// TwinCAT 3 PLC project Intecre_File
// Title: Intecre.File
// Company: Intecre Ltd
// Author: Mark Lazarides
// ProjectVersion: 1.1.0
// Description: 1.1.0 simplified interface for T_StructurePersistence 1.0.5 Increased JDOC size. 1.0.4 Fixed bug in assigning CSV separator for CsvReader 1.0.3 Clear Read and Write Success flags on struct persistence when req'd.
// ProgramVersion: 3.1.4020.4
// libraries:
//   Intecre.Utilities, * (Intecre Ltd)
//   Tc2_Standard, * (Beckhoff Automation GmbH)
//   Tc2_System, * (Beckhoff Automation GmbH)
//   Tc2_Utilities, * (Beckhoff Automation GmbH)
//   Tc3_JsonXml, * (Beckhoff Automation GmbH)
// project tree:
//   / Character.TcGVL, Param.TcGVL
//   Csv/ T_CsvFileReader.TcPOU, T_CsvFileWriter.TcPOU
//   File Bases/ E_FileBaseStates.TcDUT, T_FileReadBase.TcPOU, T_FileWriteBase.TcPOU
//   GenericFiles/ TxtFileString.TcDUT, T_TxtFileWriter.TcPOU
//   Json/ JsonDoc.TcDUT, JsonParams.TcGVL, T_StructToJsonFileWriter.TcPOU, T_StructFromJsonFileReader.TcPOU
//   Structure Persistence/ E_StructPersistenceStates.TcDUT, ST_PersistenceOptions.TcDUT, T_StructPersistence.TcPOU
//   Utilities/ E_CheckFileExistsStates.TcDUT, T_CheckFileExists.TcPOU
//   Version/ Global_Version.TcGVL

// ---- File Bases/E_FileBaseStates.TcDUT
TYPE E_FileBaseStates :
(
	WaitForStart,
	OpenFile,
	WaitForOpenComplete,
	SeekEnd,
	WaitForSeekEndComplete,
	GetSize,
	WaitForGetSizeComplete,
	SeekStart,
	WaitForSeekStartComplete,
	CreateBuffer,
	ReadFromFile,
	ReadFromFileComplete,
	WriteToFile,
	WriteToFileComplete,
	CloseFile,
	WaitForCloseComplete,
	FinishAndCleanup ) INT := WaitForStart;
END_TYPE

// ---- GenericFiles/TxtFileString.TcDUT
TYPE TxtFileString : STRING(Param.TXT_FILE_MAX_STRING_LENGTH); END_TYPE

// ---- Json/JsonDoc.TcDUT
TYPE JsonDoc : STRING( JsonParams.JSON_DOC_SIZE ); END_TYPE

// ---- Structure Persistence/E_StructPersistenceStates.TcDUT
{attribute 'qualified_only'}
{attribute 'strict'}
TYPE E_StructPersistenceStates :
(
	None,
	Initialise,
	Wait,
	ReadFromFile,
	WaitForReadComplete,
	WriteToFile,
	WaitForWriteComplete,
	Finished
);
END_TYPE

// ---- Structure Persistence/ST_PersistenceOptions.TcDUT
TYPE ST_PersistenceOptions :
STRUCT
	AddressOfStruct : PVOID;
	SizeOfStruct : UDINT;
	NameOfStructureType : STRING; // eg ST_Recipe; NOT the instance name!
	FilePath : STRING; // location to store this
	CreateFileIfDoesntExist : BOOL := TRUE; // if read fails, try a write.
	AutoWriteOnDifference : BOOL := TRUE; // if difference between
	AutoWriteCheckTime : TIME := T#2M; // how often to check for difference
	AutoWriteDebounceTime : TIME := T#30S; // time since last change to write file
END_STRUCT
END_TYPE

// ---- Utilities/E_CheckFileExistsStates.TcDUT
{attribute 'qualified_only'}
{attribute 'strict'}
TYPE E_CheckFileExistsStates :
(	
	WaitForStart,
	WaitForOpenResult,
	CloseIfOpened
);
END_TYPE

// ---- Character.TcGVL
VAR_GLOBAL CONSTANT
	CARRIAGE_RETURN : BYTE := 16#D;
	LINE_FEED : BYTE := 16#A;
	ASCI_SEMI_COLON : BYTE := 16#3B;
	ASCI_COMMA		: BYTE := 16#2C;
END_VAR

// ---- Json/JsonParams.TcGVL
{attribute 'qualified_only'}
VAR_GLOBAL CONSTANT
	JSON_DOC_SIZE : UDINT := 10000; // make this large enough for your largest structure. Add at least 20% to the byte size to account for json syntax.
END_VAR

// ---- Param.TcGVL
{attribute 'qualified_only'}
VAR_GLOBAL CONSTANT
	TXT_FILE_MAX_STRING_LENGTH : UDINT := 300;
END_VAR

// ---- Version/Global_Version.TcGVL
{attribute 'TcGenerated'}
{attribute 'no-analysis'}
{attribute 'linkalways'}
// This function has been automatically generated from the project information.
VAR_GLOBAL CONSTANT
	{attribute 'const_non_replaced'}
	stLibVersion_Intecre_File : ST_LibVersion := (iMajor := 1, iMinor := 1, iBuild := 0, iRevision := 0, nFlags := 0, sVersion := '1.1.0');
END_VAR

// ---- Csv/T_CsvFileReader.TcPOU
// Usage:
// Call instance (i.e. ofbCsvRead();) every scan while waiting for operations to complete.
// SetFileParams() Set the File directory and separator variable. 
// GetFile() Get the File.
// #various props: Observe the properties to see whether it passed the file checks.
// NextField() Next through the fields of the CSV. 
// #sField, Row, Column: Use properties to access values, using row and column.
FUNCTION_BLOCK T_CsvFileReader
VAR
// state vars.
	filePath : Tc2_Utilities.T_MaxString; // filepath
	firstField : BOOL;
	newRow : BOOL;
	
// backing properties	
	_Row : UINT;(* Row number (record) *)
	_Column : UINT;(* Column number (record field) *)
	_Field : Tc2_Utilities.T_MaxString; // Field in current Row and column
	
// Objects	
	fileRead : T_FileReadBase;(* Writes one record (line) *)
	csvReader : Tc2_Utilities.FB_CSVMemBufferReader; // read bits
	
END_VAR

fileRead();

{attribute 'monitoring' := 'call'}
PROPERTY PUBLIC Busy : BOOL
GET
Busy := fileRead.Busy;
END_GET
END_PROPERTY

PROPERTY PUBLIC Column : UINT
GET
Column := _Column;
END_GET
END_PROPERTY

{attribute 'monitoring' := 'call'}
PROPERTY PUBLIC Eof : BOOL
GET
Eof := ReadyForParsing AND NOT csvReader.bOk AND NOT firstField;
END_GET
END_PROPERTY

{attribute 'monitoring' := 'call'}
PROPERTY PUBLIC Error : BOOL
GET
Error := fileRead.Error;
END_GET
END_PROPERTY

{attribute 'monitoring' := 'call'}
PROPERTY PUBLIC ErrorId : UDINT
GET
ErrorId := fileRead.ErrorId;
END_GET
END_PROPERTY

PROPERTY PUBLIC Field : String
GET
Field := _Field;
END_GET
END_PROPERTY

PROPERTY PUBLIC FileExists : BOOL
GET
FileExists := fileRead.FileExists;
END_GET
END_PROPERTY

METHOD PUBLIC GetFile
fileRead.StartRead();
fileRead();
_Column := 0;
_Row := 0;
_Field := '';
firstField := TRUE;
newRow := FALSE;
END_METHOD

METHOD PRIVATE incrementRowAndColumn
IF newRow THEN // if it's a new row (which we know from last time)
	
	newRow := FALSE;
	_Row := _Row + 1;
	_Column := 0;
	
ELSE
	// if it's not the first read, advance column.
	IF (csvReader.eCmd = Tc2_Utilities.eEnumCmd_First) THEN
		_Column := 0;
		_Row := 0;
	ELSE
		_Column := _Column + 1;
	END_IF
	
END_IF
END_METHOD

METHOD PUBLIC NextField// gets next field
IF firstField THEN
	firstField := FALSE;
	csvReader.eCmd :=  Tc2_Utilities.E_EnumCmdType.eEnumCmd_First;
ELSE
	csvReader.eCmd :=  Tc2_Utilities.E_EnumCmdType.eEnumCmd_Next;
END_IF

processCsvReader();

// increment the column and row if necessary.
IF csvReader.bOk THEN
	incrementRowAndColumn();
	
END_IF

// increment the row number next call if necessary.
IF csvReader.bOk AND csvReader.bCRLF THEN
	newRow := TRUE;
END_IF
END_METHOD

METHOD PRIVATE processCsvReader 
// used in NextField();
csvReader(
	pBuffer:= fileRead.DataBuffer,
	cbBuffer:= fileRead.DataLength,
	getValue=> _Field);
END_METHOD

{attribute 'monitoring' := 'call'}
PROPERTY PUBLIC ReadyForParsing : BOOL
GET
ReadyForParsing := fileRead.Done;
END_GET
END_PROPERTY

PROPERTY PUBLIC Row : UINT
GET
Row := _Row;
END_GET
END_PROPERTY

METHOD PUBLIC SetFileParams
VAR_INPUT
	FilePath : Tc2_Utilities.T_MaxString;
	Separator: BYTE; // Updates TC Utilities Global_Variables DEFAULT_CSV_FIELD_SEP
END_VAR
// THIS^ references the base object properties
THIS^.filePath := FilePath; // for debug only.

fileRead.SetFilePath(FilePath := FilePath);

// Validate separator.
IF Separator = ASCI_SEMI_COLON THEN
	Tc2_Utilities.DEFAULT_CSV_FIELD_SEP := ASCI_SEMI_COLON;
	
ELSIF Separator = ASCI_COMMA THEN
	Tc2_Utilities.DEFAULT_CSV_FIELD_SEP := ASCI_COMMA;
	
ELSE
	Tc2_Utilities.DEFAULT_CSV_FIELD_SEP := ASCI_SEMI_COLON;
	
END_IF
END_METHOD

END_FUNCTION_BLOCK

// ---- File Bases/T_FileReadBase.TcPOU
(*Usage:
 N.B. FILE BUFFER IS STORED IN THIS OBJECT, IN MEMORY.  DO NOT DO ACCESS ANOTHER FILE
 		WITH THIS BLOCK UNTIL YOU HAVE FINISHED WITH IT.
 		IF YOU WANT TO EXTEND THE LIFE OF THIS BUFFFER, CREATE A NEW ONE ELSEWHERE AND MEMCPY INTO IT!
 Call instance (i.e. FileRead();) every scan while waiting for operations to complete.
 SetFilePath()
 [OPTIONAL] StartCheckFileExists(); . Only recall if necessary (i.e. long time between file path set)
  
 StartRead();

 IF BufferAvailable
 use address and size indicated by DataBuffer and DataLength.
*)

FUNCTION_BLOCK INTERNAL T_FileReadBase
VAR
// backing properties
	_FilePath : Tc2_Utilities.T_MaxString;
	_Start : BOOL;
	_Busy : BOOL;
	_Done : BOOL;
	_Error : BOOL;
	_ErrorId : UDINT;
	_Read : BOOL; // if true, reads the file.
	_FileExists: BOOL; 
	_DataBuffer : POINTER TO BYTE; // remaining data (i.e. crc is stripped).
	_DataLength : UDINT;

// Function Block Objects
	FileOpen : FB_FileOpen; // Opens file 
	FileClose : FB_FileClose; // Closes file
	FileSeek : FB_FileSeek; // Move pointer to file position.
	FileTell	: FB_FileTell; // get file information.
	FileRead	: FB_FileRead; // read from file.
	
// Vars
	CheckFileExists : BOOL;		// when set true, check the file exists.
	FileHandle : UINT;			// file handle
	FileBufferSize : UDINT;			// size of file in bytes
	FileBuffer : POINTER TO BYTE; // holds file contents

// State Enum
	State : E_FileBaseStates := E_FileBaseStates.WaitForStart;
	
END_VAR

CASE State OF
	
	E_FileBaseStates.WaitForStart:	
		
		_Busy := FALSE;
		
		IF _Start THEN
			_Start := FALSE;
			_Busy := TRUE;
			_Done := FALSE;
			_Error := FALSE;
			_ErrorId := E_AdsErr.NOERR;
			FileHandle := 0;
			State := OpenFile;
			
			// delete pointer if it previously exists. 
			IF FileBuffer > 0 THEN 
				__DELETE(FileBuffer);
			END_IF
			
		END_IF

	E_FileBaseStates.OpenFile:
	
		FileOpen(bExecute := FALSE);
		
		FileOpen( 
			sNetId 		:= '', 
			sPathName 	:= _FilePath,
			nMode 		:= FOPEN_MODEREAD OR FOPEN_MODEBINARY, // Binary uses CRLF.
			bExecute 	:= TRUE);
		// Next Step
		State := WaitForOpenComplete;

	E_FileBaseStates.WaitForOpenComplete:
	
		FileOpen(bExecute	:= FALSE,
					hFile 		=> FileHandle,
					bError 		=> _Error,
					nErrId 		=> _ErrorId);
		
		IF NOT FileOpen.bBusy THEN
			_FileExists := NOT(_ErrorId = E_AdsErr.DEVICE_NOTFOUND); // check whether file exists.
			
			IF CheckFileExists THEN	
				// if checking whether a file exists, suppress error
				CheckFileExists := FALSE;
				_Error := FALSE;
				_ErrorId := 0;
				State := FinishAndCleanup;
				
			ELSE
				State := SEL(_Error, SeekEnd, FinishAndCleanup);
			END_IF
			
		END_IF

	E_FileBaseStates.SeekEnd:
	
		// move file pointer to end of file.
		FileSeek(bExecute := FALSE);
		
	 	FileSeek(
            sNetId		:= '', 
            hFile		:= FileHandle, 
            nSeekPos	:= 0, 
            eOrigin		:= E_SeekOrigin.SEEK_END, 
            bExecute	:= TRUE);
			
		State := WaitForSeekEndComplete;
			
	E_FileBaseStates.WaitForSeekEndComplete:
	
		FileSeek(bExecute	:= FALSE,
					bError 		=> _Error,
					nErrId 		=> _ErrorId);
		
		IF NOT FileSeek.bBusy THEN
			State := SEL(_Error, GetSize, FinishAndCleanup);
		END_IF
	
	E_FileBaseStates.GetSize:
	
		// As file pointer is at the end of the file, we can find size.
		FileTell(bExecute := FALSE);
		
		FileTell(
            sNetId		:= '', 
            hFile		:= FileHandle, 
            bExecute	:= TRUE, 
            tTimeout	:= );
		
		State := WaitForGetSizeComplete;
	
	E_FileBaseStates.WaitForGetSizeComplete:
	
		FileTell(bExecute 	:= FALSE,
					bError		=> _Error, 
					nErrId		=> _ErrorId, 
					nSeekPos	=> );
		
		IF NOT FileTell.bBusy THEN
			IF _Error THEN
				State :=  FinishAndCleanup;
			ELSE
				FileBufferSize := DINT_TO_UDINT(FileTell.nSeekPos);
				State := SeekStart;
			END_IF
	
		END_IF
	
	E_FileBaseStates.SeekStart:
	
		// move file pointer to end of file.
		FileSeek(bExecute := FALSE);
		
	 	FileSeek(
            sNetId		:= '', 
            hFile		:= FileHandle, 
            nSeekPos	:= 0, 
            eOrigin		:= E_SeekOrigin.SEEK_SET, 
            bExecute	:= TRUE);
			
		State := WaitForSeekStartComplete;
	
	E_FileBaseStates.WaitForSeekStartComplete:
	
		FileSeek(bExecute 	:= FALSE,
					bError 		=> _Error,
					nErrId 		=> _ErrorId);
		
		IF NOT FileSeek.bBusy THEN
			State := SEL(_Error, CreateBuffer, FinishAndCleanup);
		END_IF
	
	E_FileBaseStates.CreateBuffer:
	
		// create the buffer
		FileBuffer := __NEW(BYTE, FileBufferSize);
		
		IF FileBuffer > 0 THEN // if successfull
			State := ReadFromFile;
			
		ELSE // create buffer failed.
			_Error 	:= TRUE;
			_ErrorId 	:= 1802; // Out of memory
			State 		:= FinishAndCleanup;
			
		END_IF

	E_FileBaseStates.ReadFromFile:
	
		FileRead(bExecute := FALSE);
		
		FileRead(
            sNetId 		:= '', 
            hFile 		:= FileHandle, 
            pReadBuff 	:= FileBuffer, 
            cbReadLen 	:= FileBufferSize, 
            bExecute 	:= TRUE, 
            tTimeout 	:= );
			
		State := ReadFromFileComplete;
		
	E_FileBaseStates.ReadFromFileComplete:
	
		FileRead(bExecute := FALSE, 
					bError 		=> _Error, 
					nErrId 		=> _ErrorId);
		
		IF NOT FileRead.bBusy THEN
			State := SEL(_Error, CloseFile, FinishAndCleanup);
		END_IF
		
	E_FileBaseStates.CloseFile:	
	
		FileClose(bExecute := FALSE);
		
		FileClose(
			sNetId 		:= '',
			hFile 		:= FileHandle, 
			bExecute 	:= TRUE);
			
		// Next Step
		State := WaitForCloseComplete;

	E_FileBaseStates.WaitForCloseComplete:
	
		FileClose(bExecute := FALSE,
					bError 		=> _Error,
					nErrId 		=> _ErrorId);
					
		IF NOT FileClose.bBusy THEN
			FileHandle := 0;
			State := FinishAndCleanup;
		END_IF

	E_FileBaseStates.FinishAndCleanup: 
		
		_Done := TRUE;
		IF NOT _error THEN
			storeDataBufferAddressAndSizeIfValid();
		END_IF
		State := SEL(FileHandle <> 0, WaitForStart, CloseFile);
		
	ELSE // Error if we get here. Tidy up if we do.
		
		F_LogError(
			CONCAT('Illegal State request in FB_FileBase. Requested State: ', TO_STRING(State))
			);
		State := FinishAndCleanup; 

END_CASE

{attribute 'monitoring' := 'call'}
PROPERTY PUBLIC BufferAvailable : BOOL
GET
BufferAvailable := _DataBuffer > 0 AND_THEN _DataLength > 0;
END_GET
END_PROPERTY

{attribute 'monitoring' := 'call'}
PROPERTY PUBLIC Busy : BOOL
GET
Busy := _Busy;
END_GET
END_PROPERTY

{attribute 'monitoring' := 'call'}
PROPERTY PUBLIC DataBuffer : POINTER TO BYTE
GET
DataBuffer := _DataBuffer;
END_GET
END_PROPERTY

{attribute 'monitoring' := 'call'}
PROPERTY PUBLIC DataLength : UDINT
GET
DataLength := _DataLength;
END_GET
END_PROPERTY

{attribute 'monitoring' := 'call'}
PROPERTY PUBLIC Done : BOOL
GET
Done := _Done;
END_GET
END_PROPERTY

PROPERTY PUBLIC Error : BOOL
GET
Error := _Error;
END_GET
END_PROPERTY

{attribute 'monitoring' := 'call'}
PROPERTY PUBLIC ErrorId : UDINT
GET
ErrorId := _ErrorId;
END_GET
END_PROPERTY

METHOD FB_exit : BOOL
VAR_INPUT
	bInCopyCode : BOOL; // if TRUE, the exit method is called for exiting an instance that is copied afterwards (online change).
END_VAR
IF FileBuffer > 0 THEN
	__DELETE(FileBuffer);
END_IF
END_METHOD

{attribute 'monitoring' := 'call'}
PROPERTY PUBLIC FileExists : BOOL
GET
FileExists := _FileExists;
END_GET
END_PROPERTY

METHOD PUBLIC SetFilePath : BOOL
VAR_INPUT
	FilePath : Tc2_Utilities.T_MaxString;
END_VAR
IF State = WaitForStart THEN
	_FilePath := FilePath;
	SetFilePath := TRUE;
ELSE
	SetFilePath := FALSE;
END_IF
END_METHOD

METHOD PUBLIC StartCheckFileExists : BOOL
IF State = WaitForStart THEN
	CheckFileExists := TRUE;
	_Start := TRUE;
	StartCheckFileExists := TRUE;
ELSE
	StartCheckFileExists := FALSE;
END_IF
END_METHOD

METHOD PUBLIC StartRead : BOOL
//validate start is possible
IF State = WaitForStart THEN
	_Start := TRUE;
	_Read	:= TRUE;
END_IF

StartRead := _Start;
END_METHOD

METHOD PRIVATE storeDataBufferAddressAndSizeIfValid
_DataBuffer := FileBuffer;
_DataLength := FileBufferSize;
END_METHOD

END_FUNCTION_BLOCK

// ---- Csv/T_CsvFileWriter.TcPOU
// Usage:
// Call instance (i.e. ofbCsvRead();) every scan while waiting for operations to complete.
// SetFileParams() Set the File directory and separator variable. 
// GetFile() Get the File.
// #various props: Observe the properties to see whether it passed the file checks.
// NextField() Next through the fields of the CSV. 
// #sField, Row, Column: Use properties to access values, using row and column.
FUNCTION_BLOCK T_CsvFileWriter
VAR
// state vars.
	filePath : Tc2_Utilities.T_MaxString; // filepath
	
// backing properties	
	_Row : UINT; // current Row number (zero indexed)
	_Column : UINT; // current Column number (zero indexed)
	_Error : BOOL;
	_ErrorId : UDINT; // E_AdsErr
	
// Objects	
	fileWrite : T_FileWriteBase;(* Writes one record (line) *)
	
END_VAR

fileWrite();

METHOD PUBLIC AddStringField// Add Field. Adds CSV separator to previous field, if it exists
VAR_INPUT 
	sFieldString : STRING; 
END_VAR

VAR_INST
	sFieldStringLocal : STRING; // This has a valid memory address (inputs dont)
END_VAR
sFieldStringLocal := sFieldString;
// append separator to previous field if not first field
IF _Column > 0 THEN 
	
	fileWrite.AppendToBuffer(
		pDataForBuffer := ADR(Tc2_Utilities.DEFAULT_CSV_FIELD_SEP),
		DataLength := SIZEOF(Tc2_Utilities.DEFAULT_CSV_FIELD_SEP)
	);	

	IF Error THEN // Error looks at FileWrite.Error
		RETURN;
	END_IF
	
END_IF

// Add string.
fileWrite.AppendToBuffer(
	pDataForBuffer := ADR(sFieldStringLocal),
	DataLength := INT_TO_UDINT(LEN(sFieldString))
);

IF Error THEN // Error looks at FileWrite.Error
	RETURN;
END_IF

_Column := _Column + 1;
END_METHOD

{attribute 'monitoring' := 'call'}
PROPERTY PUBLIC BufferClear : BOOL // ready for first entry after ResetWriteBuffer
GET
BufferClear := fileWrite.BufferClear;
END_GET
END_PROPERTY

{attribute 'monitoring' := 'call'}
PROPERTY PUBLIC Busy : BOOL
GET
Busy := fileWrite.Busy;
END_GET
END_PROPERTY

METHOD PUBLIC ClearBuffer : BOOL // Clears the buffer for first write.
ClearBuffer := fileWrite.ClearWriteBuffer();
_Error := fileWrite.Error;
_ErrorId := fileWrite.ErrorId;

_Column := 0;
_Row := 0;
END_METHOD

PROPERTY PUBLIC Column : UINT
GET
Column := _Column;
END_GET
END_PROPERTY

{attribute 'monitoring' := 'call'}
PROPERTY PUBLIC Done : BOOL
GET
Done := fileWrite.Done;
END_GET
END_PROPERTY

{attribute 'monitoring' := 'call'}
PROPERTY PUBLIC Error : BOOL
GET
_Error := fileWrite.Error;
Error := _Error;
END_GET
END_PROPERTY

{attribute 'monitoring' := 'call'}
PROPERTY PUBLIC ErrorId : UDINT
GET
_ErrorId := fileWrite.ErrorId;
ErrorId := _ErrorId;
END_GET
END_PROPERTY

METHOD PUBLIC NewLine // Make a New Line in the File
VAR_INST
	tempByte : BYTE;
END_VAR
VAR CONSTANT
	CARRIAGE_RETURN : BYTE := 16#D;
	LINE_FEED : BYTE := 16#A;
END_VAR
// load up CR.
tempByte := CARRIAGE_RETURN;

//Write.
fileWrite.AppendToBuffer(
		pDataForBuffer := ADR(tempByte),
		DataLength := SIZEOF(tempByte)
	);

// check for errors
IF Error THEN // Error looks at FileWrite.Error
	RETURN;
END_IF

// load up LF.
tempByte := LINE_FEED;

//Write.
fileWrite.AppendToBuffer(
		pDataForBuffer := ADR(tempByte),
		DataLength := SIZEOF(tempByte)
	);	

// check for errors
IF Error THEN // Error looks at FileWrite.Error
	RETURN;
END_IF

_Row := _Row + 1;
_Column := 0;
END_METHOD

PROPERTY PUBLIC Row : UINT
GET
Row := _Row;
END_GET
END_PROPERTY

METHOD SetFileOpenMode
VAR_INPUT
	Append : BOOL;  // TRUE = append, FALSE = new
END_VAR
fileWrite.SetFileOpenMode( 
	Append := Append
);
END_METHOD

METHOD PUBLIC SetFileParams
VAR_INPUT
	FilePath : Tc2_Utilities.T_MaxString;
	Separator: BYTE; // Updates TC Utilities Global_Variables DEFAULT_CSV_FIELD_SEP
END_VAR
VAR CONSTANT
	ASCI_SEMI_COLON : BYTE := 16#3B;
	ASCI_COMMA		: BYTE := 16#2C;
END_VAR
// THIS^ references the base object properties
THIS^.filePath := FilePath; // for debug only.

fileWrite.SetFilePath(FilePath := FilePath);

// Validate separator.
IF Separator = ASCI_SEMI_COLON THEN
	Tc2_Utilities.DEFAULT_CSV_FIELD_SEP := ASCI_SEMI_COLON;
	
ELSIF Separator = ASCI_COMMA THEN
	Tc2_Utilities.DEFAULT_CSV_FIELD_SEP := ASCI_COMMA;
	
ELSE
	Tc2_Utilities.DEFAULT_CSV_FIELD_SEP := ASCI_SEMI_COLON;
	
END_IF
END_METHOD

METHOD PUBLIC WriteToFile // Write Buffer to File. Calls "NewLine"() first.
// always add final CRLF.
NewLine();

fileWrite.StartWrite();
END_METHOD

END_FUNCTION_BLOCK

// ---- File Bases/T_FileWriteBase.TcPOU
(* Usage:
 N.B. THIS CLASS DOES NOT CARE ABOUT THE DATA ADDED TO THE BUFFER.
 		IF THE FINAL FILE REQUIRES LINE SEPARATORS, ADD APPRPRIATE SEPARATORS TO THE FILE AS NECESSARY.
 Call instance every scan while waiting for operations to complete.
 SetFilePath()
 ClearWriteBuffer();
 As many times as necessary: 
	AppendToBuffer();

 When finished adding to buffer.
 StartWrite();
 #various props: Observe for complete.
 *)
 
FUNCTION_BLOCK INTERNAL T_FileWriteBase
VAR
// backing properties
	_FilePath : Tc2_Utilities.T_MaxString;
	_Start : BOOL;
	_Busy : BOOL;
	_Done : BOOL;
	_Error : BOOL;
	_ErrorId : UDINT;
	_BufferClear : BOOL; // indicates reset has been called and buffer assigned.

// Function Block Objects
	FileOpen : FB_FileOpen; // Opens file
	FileClose : FB_FileClose; // Closes file
	FileWrite : FB_FileWrite; // write to file.
	
// Vars
	FileHandle : UINT;			// file handle
	
	FileBuffer : POINTER TO BYTE; // holds file contents
	FileBufferSize : UDINT;
	FileExtenderBuffer : POINTER TO BYTE; // use if buffer needs extending.

	FileOpenMode : DWORD := FOPEN_MODEWRITE OR FOPEN_MODEBINARY; // Overwrite by deafault.
	
// State Enum
	State : E_FileBaseStates := WaitForStart;
	
END_VAR
VAR CONSTANT
	FILE_OVERWRITE_MODE : DWORD := FOPEN_MODEWRITE OR FOPEN_MODEBINARY;
	FILE_APPEND_MODE : DWORD := FOPEN_MODEAPPEND OR FOPEN_MODEBINARY;	
END_VAR

CASE State OF
	
	E_FileBaseStates.WaitForStart:	
		
		_Busy := FALSE;
		
		IF _Start THEN
			_Start := FALSE;
			_Done := FALSE;
			_Error := FALSE;
			_Busy := TRUE;
			_ErrorId := E_AdsErr.NOERR;;
			FileHandle := 0;
			
			State := OpenFile;		
		END_IF

	E_FileBaseStates.OpenFile:
	
		FileOpen(bExecute := FALSE);
		
		FileOpen( 
			sNetId 		:= '', 
			sPathName 	:= _FilePath,
			nMode 		:= FileOpenMode,
			bExecute 	:= TRUE);
		// Next Step
		State := WaitForOpenComplete;

	E_FileBaseStates.WaitForOpenComplete:
	
		FileOpen(bExecute	:= FALSE,
					hFile 		=> FileHandle,
					bError 		=> _Error,
					nErrId 		=> _ErrorId);
		
		IF NOT FileOpen.bBusy THEN
			State := SEL(_Error, WriteToFile, FinishAndCleanup);		
		END_IF


	E_FileBaseStates.WriteToFile:
	
		FileWrite(bExecute := FALSE);
		
		FileWrite(
            sNetId 		:= '', 
            hFile 		:= FileHandle, 
            pWriteBuff 	:= FileBuffer, 
            cbWriteLen 	:= FileBufferSize, 
            bExecute 	:= TRUE, 
            tTimeout 	:= );
			
		State := WriteToFileComplete;
		
	E_FileBaseStates.WriteToFileComplete:
	
		FileWrite(bExecute := FALSE, 
					bError 		=> _Error, 
					nErrId 		=> _ErrorId);
		
		IF NOT FileWrite.bBusy THEN
			State := SEL(_Error, CloseFile, FinishAndCleanup);
		END_IF
		
	E_FileBaseStates.CloseFile:	
	
		FileClose(bExecute := FALSE);
		
		FileClose(
			sNetId 		:= '',
			hFile 		:= FileHandle, 
			bExecute 	:= TRUE);
			
		// Next Step
		State := WaitForCloseComplete;

	E_FileBaseStates.WaitForCloseComplete:
	
		FileClose(bExecute := FALSE,
					bError 		=> _Error,
					nErrId 		=> _ErrorId);
					
		IF NOT FileClose.bBusy THEN
			FileHandle := 0;
			State := FinishAndCleanup;
		END_IF

	E_FileBaseStates.FinishAndCleanup: 
		
		_Done := TRUE;
		State := SEL(FileHandle <> 0, WaitForStart, CloseFile);
		
	ELSE // Error if we get here. Tidy up if we do.
		
		F_LogError(
			CONCAT('Illegal State request in FB_FileWriteBase. Requested State: ', TO_STRING(State))
			);
		State := FinishAndCleanup; 

END_CASE

METHOD PUBLIC AppendToBuffer : BOOL // appends data to current line
VAR_INPUT
	pDataForBuffer : POINTER TO BYTE; // address of data start
	DataLength : UDINT; // length of data.
END_VAR
IF State = WaitForStart THEN
	
	//check valid data
	IF pDataForBuffer = 0 OR DataLength = 0 THEN
		F_LogError('Invalid data pointer passed to AppendToBuffer method.');
		RETURN;
	END_IF
	
	// append to buffer
	AppendToBuffer := 
		extendBufferSizeAndExtend(NewDataAddress := pDataForBuffer, NewDataLength := DataLength);

END_IF
END_METHOD

{attribute 'monitoring' := 'call'}
PROPERTY PUBLIC BufferClear : BOOL // ready for first entry after ResetWriteBuffer
GET
BufferClear := _BufferClear;
END_GET
END_PROPERTY

{attribute 'monitoring' := 'call'}
PROPERTY PUBLIC Busy : BOOL
GET
Busy := _Busy;
END_GET
END_PROPERTY

METHOD PUBLIC ClearWriteBuffer : BOOL // clears write buffer before adding data.
IF State = E_FileBaseStates.WaitForStart THEN
	// reset the buffer
	IF FileBuffer > 0 THEN
		__DELETE(FileBuffer);
		FileBufferSize := 0; // reset length
	END_IF
	
END_IF
END_METHOD

{attribute 'monitoring' := 'call'}
PROPERTY PUBLIC DataLength : UDINT // get size of the data in the buffer.
GET
DataLength := FileBufferSize;
END_GET
END_PROPERTY

{attribute 'monitoring' := 'call'}
PROPERTY PUBLIC Done : BOOL
GET
Done := _Done;
END_GET
END_PROPERTY

PROPERTY PUBLIC Error : BOOL
GET
Error := _Error;
END_GET
END_PROPERTY

{attribute 'monitoring' := 'call'}
PROPERTY PUBLIC ErrorId : UDINT
GET
ErrorId := _ErrorId;
END_GET
END_PROPERTY

METHOD PRIVATE extendBufferSizeAndExtend : BOOL // extends the buffer by the specified amount
VAR_INPUT
	NewDataAddress : POINTER TO BYTE;
	NewDataLength : UDINT; 
END_VAR
// make sure extension buffer empty

// If we have something in the FileBuffer, clear it down an extend it for a new buffer.
IF FileBuffer > 0 THEN
	
	IF FileExtenderBuffer > 0 THEN 
		__DELETE(FileExtenderBuffer);
	END_IF
	
	// allocate new buffer space
	FileExtenderBuffer := __NEW(BYTE, FileBufferSize);
	
	//check succesful
	IF FileExtenderBuffer = 0 THEN
		F_LogError('Out of memory trying to extend write buffer');
		_Error := TRUE;
		_ErrorId := E_AdsErr.DEVICE_NOMEMORY;
		RETURN;
	END_IF
	
	// move original data into this.
	MEMCPY(destAddr := FileExtenderBuffer, srcAddr := FileBuffer, n := FileBufferSize);
	
	// delete the old buffer
	__DELETE(FileBuffer);

END_IF

// Allocate new buffer to correct size.
FileBuffer := __NEW(BYTE, (FileBufferSize + NewDataLength));

//check for failure
IF FileBuffer = 0 THEN
	// tidy up if failed.
	__DELETE(FileExtenderBuffer); // delete this allocation.
	FileBufferSize := 0;
	F_LogError('Out of memory trying to extend write buffer');
	_Error := TRUE;
	_ErrorId := E_AdsErr.DEVICE_NOMEMORY;
	RETURN;
END_IF

// set new data to zero.
MEMSET(destAddr := FileBuffer, fillByte := 0, n := (FileBufferSize + NewDataLength));

// transfer the buffer to the original.
MEMCPY(destAddr := FileBuffer, srcAddr := FileExtenderBuffer, n := FileBufferSize);
// add the new data
MEMCPY(destAddr := ADR(FileBuffer[FileBufferSize]), srcAddr := NewDataAddress, n:= NewDataLength);
// update size.
FileBufferSize := FileBufferSize + NewDataLength;

// make sure extension buffer empty
IF FileExtenderBuffer > 0 THEN 
	__DELETE(FileExtenderBuffer);
END_IF

extendBufferSizeAndExtend := TRUE;
_BufferClear := FALSE;
END_METHOD

METHOD FB_exit : BOOL
VAR_INPUT
	bInCopyCode : BOOL; // if TRUE, the exit method is called for exiting an instance that is copied afterwards (online change).
END_VAR
// tidy up (destructor)
IF FileBuffer > 0 THEN
	__DELETE(FileBuffer);
END_IF

IF FileExtenderBuffer > 0 THEN
	__DELETE(FileExtenderBuffer);
END_IF
END_METHOD

METHOD FB_init : BOOL
VAR_INPUT
	bInitRetains : BOOL; // if TRUE, the retain variables are initialized (warm start / cold start)
	bInCopyCode : BOOL;  // if TRUE, the instance afterwards gets moved into the copy code (online change)
END_VAR
ClearWriteBuffer();
END_METHOD

METHOD SetFileOpenMode
VAR_INPUT
	Append : BOOL;  // TRUE = append, FALSE = Over write
END_VAR
FileOpenMode := SEL( Append , FILE_OVERWRITE_MODE, FILE_APPEND_MODE );
END_METHOD

METHOD PUBLIC SetFilePath : BOOL
VAR_INPUT
	FilePath : Tc2_Utilities.T_MaxString;
END_VAR
VAR_INST
	count: INT;
END_VAR
IF State = WaitForStart THEN
	_FilePath := FilePath;
	SetFilePath := TRUE;
	count := count + 1;
ELSE
	SetFilePath := FALSE;
END_IF
END_METHOD

METHOD PUBLIC StartWrite : BOOL
//validate start is possible
IF (State = WaitForStart) AND (DataLength > 0 )  THEN
	_Start := TRUE;
END_IF

StartWrite := _Start;
END_METHOD

END_FUNCTION_BLOCK

// ---- GenericFiles/T_TxtFileWriter.TcPOU
// Usage:
// Call instance every scan while waiting for operations to complete.
// SetFileParams() Set the File directory 
// GetFile() Get the File.
// #various props: Observe the properties to see whether it passed the file checks.
// NextRow()
FUNCTION_BLOCK T_TxtFileWriter
VAR
// state vars.
	filePath : Tc2_Utilities.T_MaxString; // filepath
	
// backing properties	
	_Row : UINT; // current Row number (zero indexed)
	_Error : BOOL;
	_ErrorId : UDINT; // E_AdsErr
	
// Objects	
	fileWrite : T_FileWriteBase;(* Writes one record (line) *)
	
END_VAR

fileWrite();

{attribute 'monitoring' := 'call'}
// write buffer is empty
PROPERTY PUBLIC BufferClear : BOOL
GET
BufferClear := fileWrite.BufferClear;
END_GET
END_PROPERTY

{attribute 'monitoring' := 'call'}
// file operation in progress
PROPERTY PUBLIC Busy : BOOL
GET
Busy := fileWrite.Busy;
END_GET
END_PROPERTY

// Clears the buffer (does not write to file first).
METHOD PUBLIC ClearBuffer : BOOL
ClearBuffer := fileWrite.ClearWriteBuffer();
_Error := fileWrite.Error;
_ErrorId := fileWrite.ErrorId;

_Row := 0;
END_METHOD

{attribute 'monitoring' := 'call'}
// file oepration complete
PROPERTY PUBLIC Done : BOOL
GET
Done := fileWrite.Done;
END_GET
END_PROPERTY

{attribute 'monitoring' := 'call'}
// error with buffer or file operation
PROPERTY PUBLIC Error : BOOL
GET
Error := _Error := fileWrite.Error;
END_GET
END_PROPERTY

{attribute 'monitoring' := 'call'}
// error ID
PROPERTY PUBLIC ErrorId : UDINT
GET
ErrorId := _ErrorId := fileWrite.ErrorId;
END_GET
END_PROPERTY

// Add CRLF.
METHOD PUBLIC NewLine 
VAR_INST
	tempByte : BYTE;
END_VAR
VAR CONSTANT
	CARRIAGE_RETURN : BYTE := 16#D;
	LINE_FEED : BYTE := 16#A;
END_VAR
// load up CR.
tempByte := CARRIAGE_RETURN;

//Write.
fileWrite.AppendToBuffer(
		pDataForBuffer := ADR(tempByte),
		DataLength := SIZEOF(tempByte)
	);

// check for errors
IF Error THEN // Error looks at FileWrite.Error
	RETURN;
END_IF

// load up LF.
tempByte := LINE_FEED;

//Write.
fileWrite.AppendToBuffer(
		pDataForBuffer := ADR(tempByte),
		DataLength := SIZEOF(tempByte)
	);	

// check for errors
IF Error THEN // Error looks at FileWrite.Error
	RETURN;
END_IF

_Row := _Row + 1;
END_METHOD

// current row / line number
PROPERTY PUBLIC Row : UINT
GET
Row := _Row;
END_GET
END_PROPERTY

METHOD SetFileOpenMode
VAR_INPUT
	Append : BOOL;  // TRUE = append, FALSE = new
END_VAR
fileWrite.SetFileOpenMode( 
	Append := Append
);
END_METHOD

// Set the fully scoped file path *i.e. C:/Users/TwinCAT_User/MyText.txt
METHOD PUBLIC SetFileParams
VAR_INPUT
	FilePath : Tc2_Utilities.T_MaxString;
END_VAR
THIS^.filePath := FilePath; // for debug only.

fileWrite.SetFilePath(FilePath := FilePath);
END_METHOD

// Append string to current line
METHOD PUBLIC Write
VAR_INPUT
	Entry : TxtFileString; 
END_VAR

VAR_INST
	locStr : TxtFileString; // This has a valid memory address (inputs dont)
END_VAR
locStr := Entry;

// Add string.
fileWrite.AppendToBuffer(
	pDataForBuffer := ADR(locStr),
	DataLength := INT_TO_UDINT(LEN(locStr))
);

IF Error THEN // Error looks at FileWrite.Error
	RETURN;
END_IF
END_METHOD

// Append string to current line and add CRLF
METHOD PUBLIC WriteLine
VAR_INPUT
	Entry : TxtFileString; 
END_VAR
Write( Entry );
NewLine();
END_METHOD

// Write Buffer to File.
METHOD PUBLIC WriteToFile
IF Error THEN // Error looks at FileWrite.Error
	RETURN;
END_IF

fileWrite.StartWrite();
END_METHOD

END_FUNCTION_BLOCK

// ---- Json/T_StructToJsonFileWriter.TcPOU
FUNCTION_BLOCK T_StructToJsonFileWriter EXTENDS T_NamedBase
VAR
	filePath : STRING; // fully qualified, including directory
	fileWrite : T_FileWriteBase;
	jDoc : JsonDoc;
	structureName : STRING; // i.e. 'ST_Recipe'
	pointerToStructure : PVOID; // i.e. ADR(recipe)
	sizeOfStructure : UDINT; // i.e. SIZEOF(recipe) 
	jsonWriter : FB_JsonSaxWriter;
	jsonDataTypeWriter : FB_JsonReadWriteDataType;
	_error : BOOL;
	_busy : BOOL;
	_done : BOOL;
END_VAR

fileWrite();
_error S= fileWrite.Error;
_busy := fileWrite.Busy;
_done := fileWrite.Done;

{attribute 'monitoring' := 'call' }
PROPERTY PUBLIC Busy : BOOL
GET
Busy := _busy;
END_GET
END_PROPERTY

{attribute 'monitoring' := 'call' }
PROPERTY PUBLIC Done : BOOL
GET
Done := _done;
END_GET
END_PROPERTY

{attribute 'monitoring' := 'call' }
PROPERTY PUBLIC Error : BOOL
GET
Error := _error;
END_GET
END_PROPERTY

METHOD PUBLIC Reset
fileWrite.ClearWriteBuffer();
jsonWriter.ResetDocument();
_error := FALSE;
LogDebug( 'Reset called' );
END_METHOD

METHOD PUBLIC SetFileParams
VAR_INPUT
	FilePath : Tc2_Utilities.T_MaxString;
	StructureName : STRING; // i.e. 'ST_Recipe'
	PointerToStructure : PVOID; // i.e. ADR(recipe) 
	SizeOfStructure : UDINT; // i.e. SIZEOF(recipe) 
END_VAR
THIS^.filePath := FilePath; // for debug only.
fileWrite.SetFilePath(FilePath := FilePath);

THIS^.structureName := StructureName;
THIS^.pointerToStructure := PointerToStructure; 
THIS^.sizeOfStructure := SizeOfStructure;
END_METHOD

METHOD PUBLIC WriteToFile // Attempt to write structure to file
VAR
	docSize : UDINT;
END_VAR
IF _error THEN
	LogError ( 'Cannot write to file while block is in an error state. Reset first' );
	RETURN;
	
END_IF

jsonWriter.ResetDocument();

_error S= NOT jsonDataTypeWriter.AddJsonValueFromSymbol(
						fbWriter := jsonWriter,
						sDatatype := structureName,
						nData := sizeOfStructure,
						pData := pointerToStructure	
					);
				
IF _error THEN
	LogError ( 'Error while creating json file from structure. Check argument for SetFileParams' );
	RETURN;
	
END_IF

docSize := jsonWriter.CopyDocument(
					pDoc := jDoc,
					nDoc := SIZEOF( jDoc )
				);

fileWrite.ClearWriteBuffer();

_error S= NOT fileWrite.AppendToBuffer(
						pDataForBuffer := ADR( jdoc ),
						DataLength := docSize
					);

IF _error THEN
	LogError ( 'Error while adding to write buffer. Try increasing JsonDoc size using JsonParams in library, or TC mailbox size.' );
	RETURN;
	
END_IF		
			
_error S= NOT fileWrite.StartWrite();

IF _error THEN
	LogError ( 'Error  starting file write. Try calling Reset first.' );
	RETURN;
	
END_IF
END_METHOD

END_FUNCTION_BLOCK

// ---- Json/T_StructFromJsonFileReader.TcPOU
FUNCTION_BLOCK T_StructFromJsonFileReader EXTENDS T_NamedBase
VAR
	filePath : STRING; // fully qualified, including directory
	fileRead : T_FileReadBase;
	jDoc : JsonDoc;
	structureName : STRING; // i.e. 'ST_Recipe'
	pointerToStructure : PVOID; // i.e. ADR(recipe)
	sizeOfStructure : UDINT; // i.e. SIZEOF(recipe) 
	jsonDataTypeWriter : FB_JsonReadWriteDataType;
	_error : BOOL;
	_busy : BOOL;
	_done : BOOL;
	_fileExists : BOOL;
	doneTrig : R_TRIG;
END_VAR

fileRead();
_error S= fileRead.Error;
_busy := fileRead.Busy;
_done := fileRead.Done AND fileRead.BufferAvailable;
_fileExists := fileRead.FileExists;

doneTrig( CLK := _done );

IF doneTrig.Q AND NOT _error THEN
	// clear jDoc
	MEMSET( ADR( jDoc ), 0, SIZEOF( jDoc ) );
	
	// get the data into the doc
	MEMCPY(
		destAddr := ADR( jDoc ),
		srcAddr := fileRead.DataBuffer,
		n := fileRead.DataLength
	);
	
	// conver the doc to the structure
	_error S= NOT jsonDataTypeWriter.SetSymbolFromJson(
		sJson := jDoc,
		sDatatype := structureName,
		nData := sizeOfStructure,
		pData := pointerToStructure
	);

END_IF

{attribute 'monitoring' := 'call' }
PROPERTY PUBLIC Busy : BOOL
GET
Busy := _busy;
END_GET
END_PROPERTY

{attribute 'monitoring' := 'call' }
PROPERTY PUBLIC Done : BOOL
GET
Done := _done;
END_GET
END_PROPERTY

{attribute 'monitoring' := 'call' }
PROPERTY PUBLIC Error : BOOL
GET
Error := _error;
END_GET
END_PROPERTY

{attribute 'monitoring' := 'call'}
PROPERTY PUBLIC FileExists : BOOL
GET
FileExists := _fileExists;
END_GET
END_PROPERTY

METHOD ReadFromFile // start the read.
IF _error THEN
	LogError ( 'Cannot read from file while block is in an error state. Reset first' );
	RETURN;
	
END_IF

_error S= NOT fileRead.StartRead();

IF _error THEN
	LogError ( 'ReadFromFile error, try Rest or wait until not busy' );
	RETURN;
	
END_IF
END_METHOD

METHOD PUBLIC Reset
_error := FALSE;
LogDebug( 'Reset called' );
END_METHOD

METHOD PUBLIC SetFileParams
VAR_INPUT
	FilePath : Tc2_Utilities.T_MaxString;
	StructureName : STRING; // i.e. 'ST_Recipe'
	PointerToStructure : PVOID; // i.e. ADR(recipe) 
	SizeOfStructure : UDINT; // i.e. SIZEOF(recipe) 
END_VAR
THIS^.filePath := FilePath; // for debug only.
fileRead.SetFilePath( FilePath := FilePath );

THIS^.structureName := StructureName;
THIS^.pointerToStructure := PointerToStructure; 
THIS^.sizeOfStructure := SizeOfStructure;
END_METHOD

END_FUNCTION_BLOCK

// ---- Structure Persistence/T_StructPersistence.TcPOU
FUNCTION_BLOCK T_StructPersistence
VAR_INPUT
	Options : ST_PersistenceOptions;
END_VAR
VAR_OUTPUT
	ReadSuccess : BOOL;
	WriteSuccess : BOOL;
	FileCreated : BOOL; // if the file is written without a valid file having been read first. 
END_VAR
VAR
	toFile : T_StructToJsonFileWriter;
	fromFile : T_StructFromJsonFileReader;
	lastGoodCrc : WORD; // the crc of the last file. Used for diff.
	currStructCrc, prevCheckStructCrc : WORD;
	diffCheckTimer : TON;
	diffCheckDebouncing : BOOL;
	diffDebounceTimer : TON;
	
	firstWriteSuccess : SR;
	firstSuccessTrig : R_TRIG;
	
	state : E_StructPersistenceStates;
	
END_VAR

CASE state OF
	E_StructPersistenceStates.None :
		state := E_StructPersistenceStates.Initialise;
	
	E_StructPersistenceStates.Initialise :
	
		toFile.SetFileParams(
			FilePath := Options.FilePath,
			StructureName :=	Options.NameOfStructureType,
			PointerToStructure := Options.AddressOfStruct,
			SizeOfStructure := Options.SizeOfStruct
		);
		
		fromFile.SetFileParams(
			FilePath := Options.FilePath,
			StructureName := Options.NameOfStructureType,
			PointerToStructure := Options.AddressOfStruct,
			SizeOfStructure := Options.SizeOfStruct
		);
		
		toFile.Reset();
		fromFile.Reset();
		
		state := E_StructPersistenceStates.ReadFromFile;
		
	E_StructPersistenceStates.Wait :
		; // advanced elsewhere
	
	E_StructPersistenceStates.ReadFromFile :
	
		fromFile.ReadFromFile();
		state := E_StructPersistenceStates.WaitForReadComplete;
		 
	E_StructPersistenceStates.WaitForReadComplete :
		
		ReadSuccess := fromFile.Done;
		
		IF NOT fromFile.Busy THEN
			
			IF ReadSuccess THEN 
				// record crc for diff checks	
				lastGoodCrc := getStructCrc();
				
			END_IF
			
			// if no file found, check whether to auto create (option).
			state := 
				SEL( NOT fromFile.FileExists AND Options.CreateFileIfDoesntExist, E_StructPersistenceStates.Wait, E_StructPersistenceStates.WriteToFile );	
			
			fromFile.Reset();
			
		END_IF
		
	E_StructPersistenceStates.WriteToFile :
	
		tofile.WriteToFile();
		state := E_StructPersistenceStates.WaitForWriteComplete;
		
	E_StructPersistenceStates.WaitForWriteComplete :
	
		WriteSuccess := toFile.Done;
		
		IF NOT toFile.Busy THEN
			
			IF WriteSuccess THEN
				// get the crc of the file as it's written. this allows checking for diff.			
				lastGoodCrc := getStructCrc();
				
			END_IF
			
			toFile.Reset();
			state := E_StructPersistenceStates.Wait;
			
		END_IF

END_CASE

// run file handlers
toFile();
fromFile();

firstWriteSuccess( SET1 := WriteSuccess );
firstSuccessTrig( CLK := firstWriteSuccess.Q1 );
FileCreated S= firstSuccessTrig.Q AND NOT fromFile.FileExists;

// below is auto persistence, based on the "Options" imput.

// check for difference
diffCheckTimer( 
	IN := Options.AutoWriteOnDifference AND NOT diffCheckTimer.Q AND NOT diffCheckDebouncing, 
	PT := Options.AutoWriteCheckTime
);

IF diffCheckTimer.Q THEN
	currStructCrc := getStructCrc();
	diffCheckDebouncing := ( lastGoodCrc <> currStructCrc );
	
END_IF

// once a difference has been detected, debounce changes to the struct before writing to file
diffDebounceTimer( 
	IN := diffCheckDebouncing AND NOT diffDebounceTimer.Q,
	PT := Options.AutoWriteDebounceTime
);

// when no more changes to the file, write.
IF diffDebounceTimer.Q THEN
	
 	prevCheckStructCrc := currStructCrc;
	currStructCrc := getStructCrc();
	
	// wait for struct to show no change since last debounce check
	diffCheckDebouncing := ( currStructCrc <> prevCheckStructCrc ) AND ( state = E_StructPersistenceStates.Wait );
	
	// when struct stops changing, 
	IF NOT diffCheckDebouncing THEN
		state := E_StructPersistenceStates.WriteToFile;		
		
	END_IF
	
END_IF

METHOD PRIVATE getStructCrc : WORD
getStructCrc := 
	F_DATA_TO_CRC16_CCITT(
		pData := Options.AddressOfStruct,
		cbData := Options.SizeOfStruct,
		crc := 16#FFFF // seed the CRC
	);
END_METHOD

METHOD PUBLIC ReadFromFile : BOOL
IF state <> E_StructPersistenceStates.Wait THEN
	RETURN;
END_IF

ReadFromFile := TRUE;
ReadSuccess := FALSE;
WriteSuccess := FALSE;
FileCreated := FALSE;

state := E_StructPersistenceStates.ReadFromFile;
END_METHOD

METHOD PUBLIC WriteToFile : BOOL
IF state <> E_StructPersistenceStates.Wait THEN
	RETURN;
END_IF

WriteToFile := TRUE;

ReadSuccess := FALSE;
WriteSuccess := FALSE;
FileCreated := FALSE;

state := E_StructPersistenceStates.WriteToFile;
END_METHOD

END_FUNCTION_BLOCK

// ---- Utilities/T_CheckFileExists.TcPOU
FUNCTION_BLOCK T_CheckFileExists
VAR
	fileOpen : FB_FileOpen;
	fileClose : FB_FileClose;
	
	start : BOOL;
	_fileExists : BOOL; 
	
	state : E_CheckFileExistsStates;
	
END_VAR

CASE state OF
	
	E_CheckFileExistsStates.WaitForStart : 
	
		IF start THEN
			 _fileExists := FALSE;
			 state := E_CheckFileExistsStates.WaitForOpenResult;
			 start := FALSE;
		END_IF
		
	E_CheckFileExistsStates.WaitForOpenResult : 
	
		IF NOT fileOpen.bBusy THEN
			state := SEL( fileOpen.bError, E_CheckFileExistsStates.CloseIfOpened, E_CheckFileExistsStates.WaitForStart );		
		END_IF
		
	E_CheckFileExistsStates.CloseIfOpened : 
	
		IF NOT fileClose.bBusy THEN
			state := E_CheckFileExistsStates.WaitForStart;		
		END_IF
		
END_CASE

fileOpen(
	sNetId 		:= '', 
	nMode 		:= FOPEN_MODEREAD,
	bExecute 	:= state = E_CheckFileExistsStates.WaitForOpenResult
);
	
fileClose( 
	sNetId := '', 
   hFile := fileOpen.hFile,
	bExecute := state = E_CheckFileExistsStates.CloseIfOpened
);
	
_fileExists S= state = E_CheckFileExistsStates.CloseIfOpened;

{attribute 'monitoring' := 'variable'}
PROPERTY Busy : BOOL
GET
Busy := 
	start OR ( state <> E_CheckFileExistsStates.WaitForStart );
END_GET
END_PROPERTY

METHOD Check
VAR_INPUT
	Path : STRING; // path for new file. 
END_VAR
FileOpen( 
	sPathName := Path
);

start := TRUE;
END_METHOD

{attribute 'monitoring' := 'variable'}
PROPERTY FileExists : BOOL
GET
FileExists := _fileExists AND NOT Busy;
END_GET
END_PROPERTY

END_FUNCTION_BLOCK
